{attribute addProperty BoxType "EL2564-0000-0016"}
{attribute addProperty Id "WarningBIT10.1256ErrorBIT10.1257TxPDO_ToggleBIT10.12516"}
{attribute addProperty CRC "548865613"}
{attribute addProperty SizeInBites "16"}
{attribute addProperty SizeInBytes "2"}
TYPE Status_20B7064D :
STRUCT
	{attribute 'hide'}
	reserve_1_BIT_0 : BIT;
	{attribute 'hide'}
	reserve_1_BIT_1 : BIT;
	{attribute 'hide'}
	reserve_1_BIT_2 : BIT;
	{attribute 'hide'}
	reserve_1_BIT_3 : BIT;
	{attribute 'hide'}
	reserve_1_BIT_4 : BIT;
	{attribute addProperty Name "Warning"}
	Warning : BIT;
	{attribute addProperty Name "Error"}
	Error : BIT;
	{attribute 'hide'}
	reserve_2 : BYTE;
	{attribute addProperty Name "TxPDO_Toggle"}
	TxPDO_Toggle : BIT;
END_STRUCT
END_TYPE

(* stored: Version 1.2.0.0, ProductVersion 3.1.4024.9
   DUT Status_20B7064D: Id {7315dc40-5aee-4197-bcec-5c684a506438} *)
